Omron CX-Programmer project 新工程 (CX-Programmer 9.73)

# PLC 新PLC1: CPM1(CPM1A) CPU20

## Global symbols (name address type ; comment)
0.00 BOOL  ; 急停
0.01 BOOL  ; 启动
0.03 BOOL  ; 定位
0.04 BOOL  ; 翻坯电眼
0.07 BOOL  ; 翻坯/过砖
10.01 BOOL  ; 翻坯
10.02 BOOL  ; 翻棒
10.04 BOOL  ; 前棒
12.00 BOOL  ; 允许运行
12.01 BOOL  ; 运行
5.01 BOOL  ; 启动翻棒
5.02 BOOL  ; 翻前脉冲
5.03 BOOL  ; 翻坯
5.04 BOOL  ; 定前脉冲
5.05 BOOL  ; 电眼后脉冲
CNT001 BOOL  ; 延时翻坯

## Program 新程序1 (no task)
; 以下是我设计的一个PLC示例程序，主要实现了一个釉线翻坯机系统的控制系统。我将它应用于陶瓷生产线的自动化控制，具体场景为陶瓷厂的釉料喷涂前工序。 / 系统包含启动按钮、急停按钮、定位信号、翻坯电眼和翻坯/过砖开关作为输入设备。 / 执行器包括翻坯电机、翻棒电机和前棒电机。 / 系统通过启动按钮或允许运行标志为真，且急停按钮未被按下时，设置允许运行标志；随后在允许运行标志为真时，设置运行标志。 / 急停按钮被按下时，重置允许运行标志，从而间接停止翻坯电机、翻棒电机和前棒电机，确保操作人员和设备安全。 / 在陶瓷生产线上，坯料被放置在传送带上，当翻坯电眼检测到坯料时，系统启动后续动作，并根据翻坯/过砖开关的状态分别控制翻棒电机和前棒电机。 / 若进入翻坯模式，翻坯电眼触发后首先延时80个单位时间；随后通过延时翻坯计数器计数10个单位时间，确保坯料稳定。 / 延时完成后，若定位信号为真，翻棒电机启动；翻坯电机由翻坯标志控制，其设置依赖定位信号。 / 这一机制确保翻棒电机和翻坯电机在坯料准确定位时运行，避免位置偏差影响操作。 / 若翻坯/过砖开关表示过砖模式，前棒电机启动，将坯料平稳输送至下一工序。 / 在翻坯过程中，翻棒电机的启动依赖于启动翻棒标志和运行标志为真，同时翻坯标志和翻坯/过砖开关为假，并在定位信号确认为真后运行。 / 翻坯电机由翻坯标志和允许运行标志控制，翻坯标志在定位信号确认后设置，确保动作精准。

### Section 段1

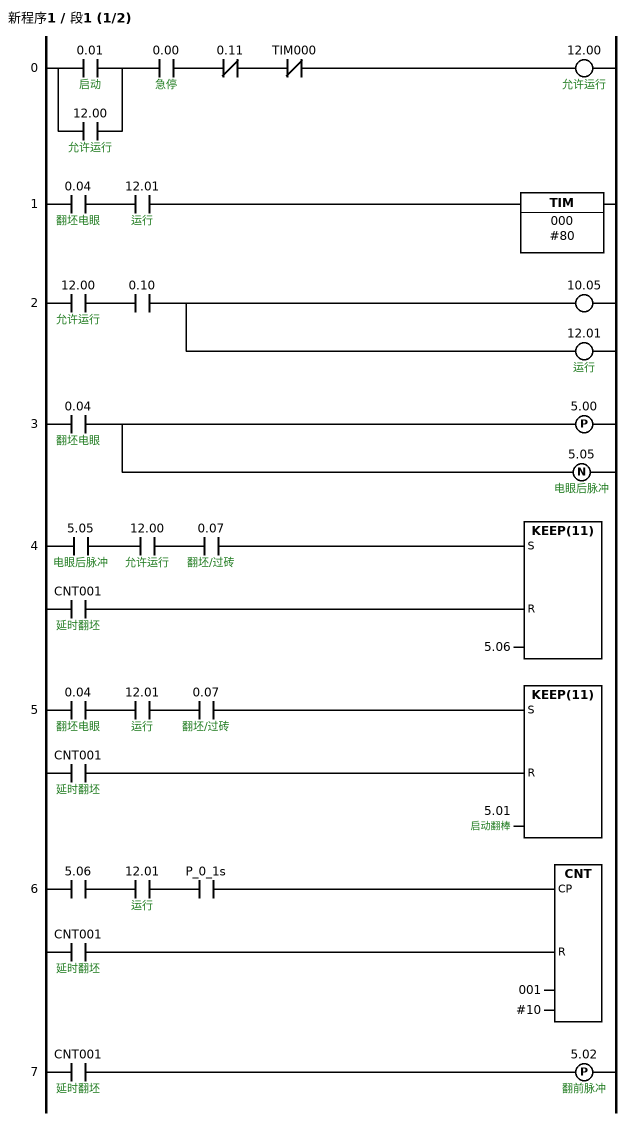
; rung 0
LD 0.01  ; 启动
OR 12.00  ; 允许运行
AND 0.00  ; 急停
ANDNOT 0.11
ANDNOT TIM000
OUT 12.00  ; 允许运行
; rung 1
LD 0.04  ; 翻坯电眼
AND 12.01  ; 运行
TIM 000 #80
; rung 2
LD 12.00  ; 允许运行
AND 0.10
OUT 10.05
OUT 12.01  ; 运行
; rung 3
LD 0.04  ; 翻坯电眼
DIFU(13) 5.00
DIFD(14) 5.05  ; 电眼后脉冲
; rung 4
LD 5.05  ; 电眼后脉冲
AND 12.00  ; 允许运行
AND 0.07  ; 翻坯/过砖
LD CNT001  ; 延时翻坯
KEEP(11) 5.06
; rung 5
LD 0.04  ; 翻坯电眼
AND 12.01  ; 运行
AND 0.07  ; 翻坯/过砖
LD CNT001  ; 延时翻坯
KEEP(11) 5.01  ; 启动翻棒
; rung 6
LD 5.06
AND 12.01  ; 运行
AND P_0_1s
LD CNT001  ; 延时翻坯
CNT 001 #10
; rung 7
LD CNT001  ; 延时翻坯
DIFU(13) 5.02  ; 翻前脉冲

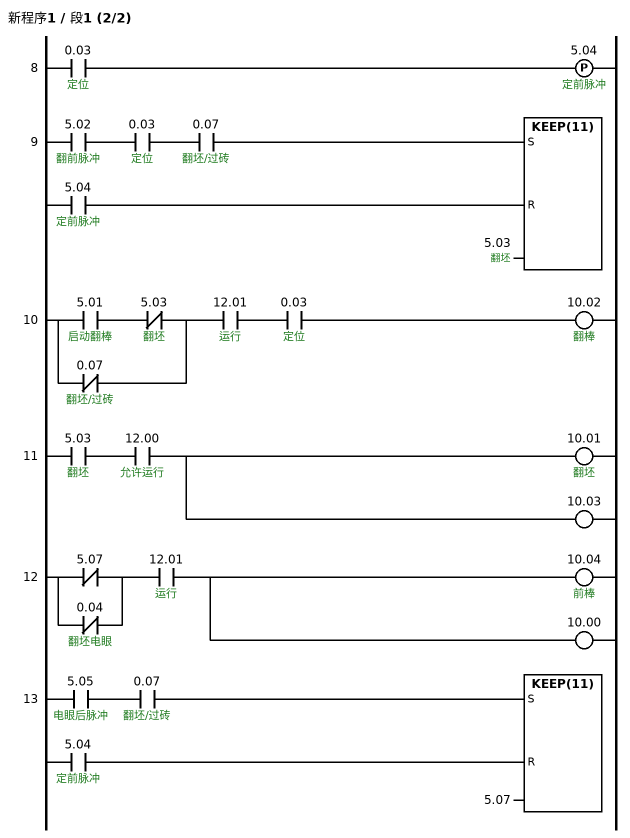
; rung 8
LD 0.03  ; 定位
DIFU(13) 5.04  ; 定前脉冲
; rung 9
LD 5.02  ; 翻前脉冲
AND 0.03  ; 定位
AND 0.07  ; 翻坯/过砖
LD 5.04  ; 定前脉冲
KEEP(11) 5.03  ; 翻坯
; rung 10
LD 5.01  ; 启动翻棒
ANDNOT 5.03  ; 翻坯
ORNOT 0.07  ; 翻坯/过砖
AND 12.01  ; 运行
AND 0.03  ; 定位
OUT 10.02  ; 翻棒
; rung 11
LD 5.03  ; 翻坯
AND 12.00  ; 允许运行
OUT 10.01  ; 翻坯
OUT 10.03
; rung 12
LDNOT 5.07
ORNOT 0.04  ; 翻坯电眼
AND 12.01  ; 运行
OUT 10.04  ; 前棒
OUT 10.00
; rung 13
LD 5.05  ; 电眼后脉冲
AND 0.07  ; 翻坯/过砖
LD 5.04  ; 定前脉冲
KEEP(11) 5.07
; rung 14
END(01)